ABB RobotStudio station: proyecto final.rspag

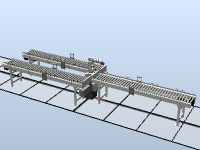
--- station ---
Station proyecto final_4 (saved by RobotStudio 6.8.8307.1040)
Controller ProyectoFinal, task T_ROB1: task frame (RAPID world) sits at (45.04, 0, 650) mm in the station
Controller ProyectoFinal
  mechanical unit ROB_1: IRB120_3_58__01, 6 joints, base frame (0, 0, 0) mm
Layout (positions relative to the parent item):
  - IRB120_3_58__01 [mechanism, from Robots\IRB120_3_58_G_01.rslib] at (45.04, 0, 650) mm; joint values [0, 0, 0, 0, 0.5236, 0] (rad or m)
  - RobotBase [part, from Descargas del Explorador\RobotBase.rslib] at (-150, -150, 0) mm
  - 400_guide [part, from Equipment\Conveyor Guide 400.rslib] at (192.48, -209.68, 0) mm
  - 400_guide_Big [part, from Equipment\Conveyor Guide 400.rslib] at (168.85, 683.15, 0) mm, rotated rx 0 ry 0 rz 180 deg
  - 400_guide_Small [part, from Equipment\Conveyor Guide 400.rslib] at (130.41, -257.14, 0) mm, rotated rx 0 ry 0 rz 180 deg
  - Big_Can [part] at (3492.94, 0, 776.65) mm
  - Little_Can [part] at (3339.79, 0, 775.69) mm
  - SmartComponent_1 [smart component]
      signals: DI Cinta1, DI Marcha, DO Sensor1Big, DO Sensor1Small, DI Cinta2Big, DI Cinta2Small, DI CogerC1Big, DI CogerC1Small, DI DejarC1Big, DI DejarC1Small, DO Sensor2Big, DO Sensor2Small, DI Cinta1S, DI Marcha1S
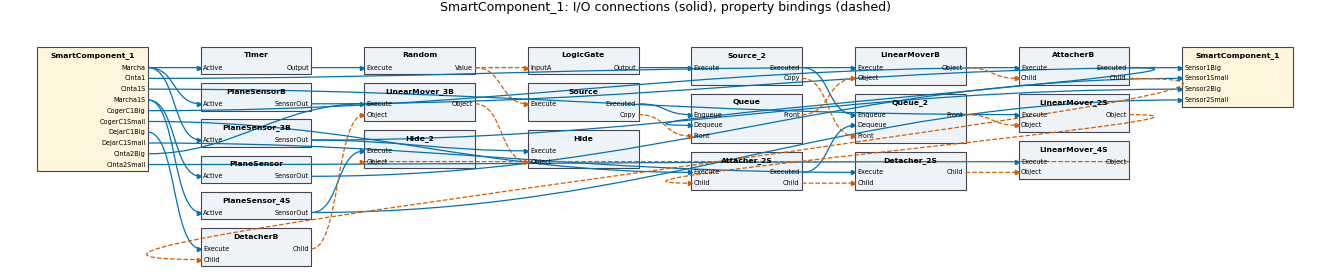
      connections:
        SmartComponent_1.Marcha -> Timer.Active
        Timer.Output -> Random.Execute
        LogicGate.Output -> Source_2.Execute
        Source.Executed -> Queue.Enqueue
        Source_2.Executed -> Queue_2.Enqueue
        SmartComponent_1.Cinta1 -> LinearMoverB.Execute
        SmartComponent_1.Cinta1S -> LinearMover_2S.Execute
        PlaneSensorB.SensorOut -> SmartComponent_1.Sensor1Big
        PlaneSensor.SensorOut -> SmartComponent_1.Sensor1Small
        SmartComponent_1.Marcha -> PlaneSensorB.Active
        SmartComponent_1.Marcha1S -> PlaneSensor.Active
        SmartComponent_1.CogerC1Big -> AttacherB.Execute
        SmartComponent_1.CogerC1Small -> Attacher_2S.Execute
        SmartComponent_1.DejarC1Big -> DetacherB.Execute
        SmartComponent_1.DejarC1Small -> Detacher_2S.Execute
        SmartComponent_1.Marcha -> PlaneSensor_3B.Active
        SmartComponent_1.Marcha1S -> PlaneSensor_4S.Active
        PlaneSensor_3B.SensorOut -> SmartComponent_1.Sensor2Big
        PlaneSensor_4S.SensorOut -> SmartComponent_1.Sensor2Small
        SmartComponent_1.Cinta2Big -> LinearMover_3B.Execute
        SmartComponent_1.Cinta2Small -> LinearMover_4S.Execute
        AttacherB.Executed -> Queue.Dequeue
        Attacher_2S.Executed -> Queue_2.Dequeue
        PlaneSensor_3B.SensorOut -> Hide.Execute
        PlaneSensor_4S.SensorOut -> Hide_2.Execute
        Random.Value => LogicGate.InputA
        Random.Value => Source.Execute
        Source.Copy => Queue.Front
        Source_2.Copy => Queue_2.Front
        Queue.Front => LinearMoverB.Object
        Queue_2.Front => LinearMover_2S.Object
        LinearMoverB.Object => AttacherB.Child
        LinearMover_2S.Object => Attacher_2S.Child
        AttacherB.Child => DetacherB.Child
        Attacher_2S.Child => Detacher_2S.Child
        DetacherB.Child => LinearMover_3B.Object
        Detacher_2S.Child => LinearMover_4S.Object
        LinearMover_3B.Object => Hide.Object
        LinearMover_4S.Object => Hide_2.Object
    - PlaneSensorB [smart component, from Components\PlaneSensor.rslib] at (395.44, -52.44, 915.91) mm, rotated rx 0 ry -90 rz 0 deg
        properties: Origin=[0 0 0]; Axis1=[0.1 0 0]; Axis2=[0 0.1 0]; SensedPart=(none)
      - _sensorPart_ [part, from Components\PlaneSensor.rslib]
    - Timer [smart component, from Components\Timer.rslib]
        properties: StartTime=0; Interval=7; Repeat=true; CurrentTime=20.088
    - Queue [smart component, from Components\Queue.rslib]
        properties: Back=(none); Front=(none); Queue=; NumberOfObjects=0
    - Queue_2 [smart component, from Components\Queue.rslib]
        properties: Back=(none); Front=(none); Queue=; NumberOfObjects=0
    - Source [smart component, from Components\Source.rslib]
        properties: Source=Big_Can; Copy=(none); Parent=(none); Position=[2.892064 0 0.776651]; Orientation=[0 0 0]; Transient=true; PhysicsBehavior=0
    - Source_2 [smart component, from Components\Source.rslib]
        properties: Source=Little_Can; Copy=(none); Parent=(none); Position=[2.753947 0 0.775688]; Orientation=[0 0 0]; Transient=true; PhysicsBehavior=0
    - LinearMoverB [smart component, from Components\LinearMover.rslib]
        properties: Object=(none); Direction=[-1 0 0]; Speed=0.8; Reference=Global; ReferenceObject=(none)
    - Random [smart component, from Components\Random.rslib]
        properties: Value=0.788703927206203; Min=0; Max=1
    - LogicGate [smart component, from Components\LogicGate.rslib]
        properties: Operator=NOT; Delay=0
    - LinearMover_2S [smart component, from Components\LinearMover.rslib]
        properties: Object=(none); Direction=[-1 0 0]; Speed=0.8; Reference=Global; ReferenceObject=(none)
    - PlaneSensor_3B [smart component, from Components\PlaneSensor.rslib] at (-2635.89, 427.82, 780.39) mm
        properties: Origin=[0 0 0]; Axis1=[0.1 0 0]; Axis2=[0 0.1 0]; SensedPart=(none)
      - _sensorPart_ [part, from Components\PlaneSensor.rslib]
    - PlaneSensor_4S [smart component, from Components\PlaneSensor.rslib] at (-2612.83, -525.9, 779.66) mm
        properties: Origin=[0 0 0]; Axis1=[0.1 0 0]; Axis2=[0 0.1 0]; SensedPart=(none)
      - _sensorPart_ [part, from Components\PlaneSensor.rslib]
    - AttacherB [smart component, from Components\Attacher.rslib]
        properties: Parent=subcionador pro; Flange=0; Child=(none); Mount=false; Offset=[0 0 0]; Orientation=[0 0 0]
    - Attacher_2S [smart component, from Components\Attacher.rslib]
        properties: Parent=subcionador pro; Flange=0; Child=(none); Mount=false; Offset=[0 0 0]; Orientation=[0 0 0]
    - DetacherB [smart component, from Components\Detacher.rslib]
        properties: Child=(none); KeepPosition=true
    - Detacher_2S [smart component, from Components\Detacher.rslib]
        properties: Child=(none); KeepPosition=true
    - LinearMover_3B [smart component, from Components\LinearMover.rslib]
        properties: Object=(none); Direction=[-1 0 0]; Speed=1.8; Reference=Global; ReferenceObject=(none)
    - LinearMover_4S [smart component, from Components\LinearMover.rslib]
        properties: Object=(none); Direction=[-1 0 0]; Speed=1.8; Reference=Global; ReferenceObject=(none)
    - PlaneSensor [smart component, from Components\PlaneSensor.rslib] at (387.44, -48.08, 820.06) mm, rotated rx 0 ry -90 rz 0 deg
        properties: Origin=[0 0 0]; Axis1=[0.1 0 0]; Axis2=[0 0.1 0]; SensedPart=(none)
      - _sensorPart_ [part, from Components\PlaneSensor.rslib]
    - Hide [smart component, from Components\Hide.rslib]
        properties: Object=(none)
    - Hide_2 [smart component, from Components\Hide.rslib]
        properties: Object=(none)
  - subcionador pro [mechanism, from Videos\subcionador pro.rslib] at (409.39, 0, 1244) mm, rotated rx 180 ry 60 rz 180 deg
Attachment: subcionador pro is attached to IRB120_3_58__01 / Link6
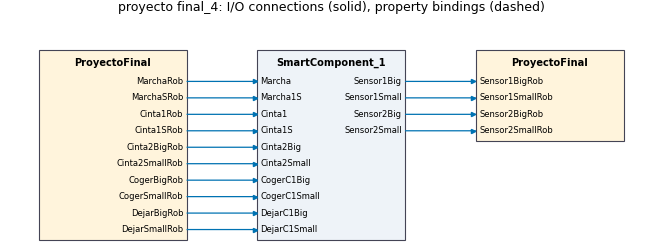
Station logic (signal -> signal, property => property):
  ProyectoFinal.MarchaRob -> SmartComponent_1.Marcha
  ProyectoFinal.MarchaSRob -> SmartComponent_1.Marcha1S
  ProyectoFinal.Cinta1Rob -> SmartComponent_1.Cinta1
  ProyectoFinal.Cinta1SRob -> SmartComponent_1.Cinta1S
  SmartComponent_1.Sensor1Big -> ProyectoFinal.Sensor1BigRob
  SmartComponent_1.Sensor1Small -> ProyectoFinal.Sensor1SmallRob
  ProyectoFinal.Cinta2BigRob -> SmartComponent_1.Cinta2Big
  ProyectoFinal.Cinta2SmallRob -> SmartComponent_1.Cinta2Small
  ProyectoFinal.CogerBigRob -> SmartComponent_1.CogerC1Big
  ProyectoFinal.CogerSmallRob -> SmartComponent_1.CogerC1Small
  ProyectoFinal.DejarBigRob -> SmartComponent_1.DejarC1Big
  ProyectoFinal.DejarSmallRob -> SmartComponent_1.DejarC1Small
  SmartComponent_1.Sensor2Big -> ProyectoFinal.Sensor2BigRob
  SmartComponent_1.Sensor2Small -> ProyectoFinal.Sensor2SmallRob
Targets, tools, work objects and paths stored in the station and not in the controller backup, written as RAPID:
! task T_ROB1
MODULE Module1
  PROC pieza()
    robotSmall;
    sensar1;
  ENDPROC
  PROC cicle()
    SetDO CogerBigRob,0;
    SetDO DejarBigRob,0;
    SetDO CogerSmallRob,0;
    SetDO DejarSmallRob,0;
    SetDO MarchaRob,1;
    SetDO MarchaSRob,1;
    SetDO Cinta1Rob,1;
    SetDO Cinta1SRob,1;
    SetDO Cinta2BigRob,0;
    SetDO Cinta2SmallRob,0;
    WaitDI Sensor1SmallRob,1;
    SetDO Cinta1Rob,0;
    SetDO Cinta1SRob,0;
    piezas;
  ENDPROC
  PROC sensar()
    cicle;
    cicle;
  ENDPROC
ENDMODULE


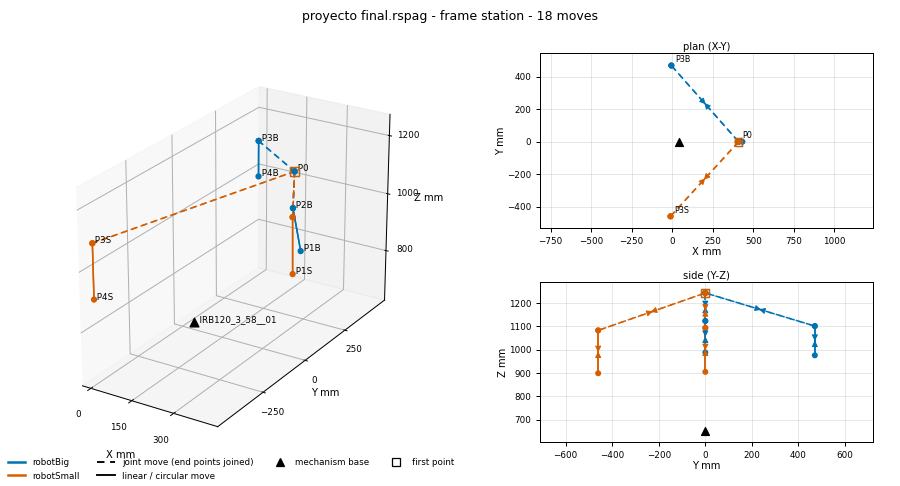
[picture p0: tool path of proyecto final.rspag in frame station, 18 of 18 moves have a stored position in this frame; points joined in program order, loops and branches not executed]
--- Backups/ProyectoFinal/RAPID/TASK1/PROGMOD/CalibData.mod ---
MODULE CalibData
ENDMODULE

--- Backups/ProyectoFinal/RAPID/TASK1/PROGMOD/Module1.mod ---
MODULE Module1
    CONST robtarget P0:=[[364.353829072,0,594],[0.5,0,0.866025404,0],[0,0,0,0],[9E+09,9E+09,9E+09,9E+09,9E+09,9E+09]];
    CONST robtarget P2B:=[[360.022653153,0,473.726196092],[0,0,1,0],[0,0,0,0],[9E+09,9E+09,9E+09,9E+09,9E+09,9E+09]];
    CONST robtarget P1B:=[[388.755601806,0,338.420809037],[0,0,1,0],[0,0,0,0],[9E+09,9E+09,9E+09,9E+09,9E+09,9E+09]];
    CONST robtarget P3B:=[[-50.206591399,470.402076052,451.620152637],[0,0,1,0],[0,0,0,0],[9E+09,9E+09,9E+09,9E+09,9E+09,9E+09]];
    CONST robtarget P4B:=[[-50.206591399,470.402076052,325.966309799],[0,0,1,0],[0,0,0,0],[9E+09,9E+09,9E+09,9E+09,9E+09,9E+09]];
    CONST robtarget P2S:=[[359.130975003,0,443.778021736],[0,0,1,0],[0,0,0,0],[9E+09,9E+09,9E+09,9E+09,9E+09,9E+09]];
    CONST robtarget P1S:=[[361.332509941,0,254.842738956],[0,0,1,0],[0,0,0,0],[9E+09,9E+09,9E+09,9E+09,9E+09,9E+09]];
    CONST robtarget P3S:=[[-55.454860484,-460.39542717,433.082453731],[0,0,1,0],[-2,0,-2,0],[9E+09,9E+09,9E+09,9E+09,9E+09,9E+09]];
    CONST robtarget P4S:=[[-55.454860484,-460.39542717,248.927934739],[0,0,1,0],[-2,0,-2,0],[9E+09,9E+09,9E+09,9E+09,9E+09,9E+09]];
	PERS tooldata subcionador_pro:=[TRUE,[[0,0,0],[1,0,0,0]],[2,[0,0,1],[1,0,0,0],0,0,0]];
    !***********************************************************
    !
    ! Module:  Module1
    !
    ! Description:
    !   <Pick and Place de dos diferentes latas>
    !
    ! Author: Kenneth
    !
    ! Version: 1.0
    !
    !***********************************************************


    !***********************************************************
    !
    ! Procedure main
    !
    !   This is the entry point of your program
    !
    !***********************************************************
    PROC main()
        !Aqui pongo las señales de agarrar y soltar las latas en 0, así cada vez que se inicia, empiezan en 0
        SetDO CogerBigRob,0;
        SetDO DejarBigRob,0;
        SetDO CogerSmallRob,0;
        SetDO DejarSmallRob,0;
        !Aquí pongo en marcha la cinta, son dos porque para evitar cualquier error hice que cada lata actuara
        !como si se movieran en cintas diferentes
        SetDO MarchaRob,1;
        SetDO MarchaSRob,1;
        SetDO Cinta1Rob,1;
        SetDO Cinta1SRob,1;
        SetDO Cinta2BigRob,0;
        SetDO Cinta2SmallRob,0;
        !Apenas el sensor que tiene contacto con los dos tipos de latas recibe una señal, para la cinta para
        !realizar la función piezas
        WaitDI Sensor1SmallRob,1;
        SetDO Cinta1Rob,0;
        SetDO Cinta1SRob,0;
        piezas;
    ENDPROC
    PROC robotBig()
        !Trayectoria para las latas grandes
        MoveJ P0,v1000,z100,subcionador_pro\WObj:=wobj0;
        MoveJ P2B,v1000,z100,subcionador_pro\WObj:=wobj0;
        MoveL P1B,v1000,fine,subcionador_pro\WObj:=wobj0;
        SetDO CogerBigRob,1;
        MoveL P2B,v1000,z100,subcionador_pro\WObj:=wobj0;
        MoveJ P0,v1000,z100,subcionador_pro\WObj:=wobj0;
        MoveJ P3B,v1000,z100,subcionador_pro\WObj:=wobj0;
        MoveL P4B,v1000,fine,subcionador_pro\WObj:=wobj0;
        SetDO DejarBigRob,1;
        SetDO Cinta2BigRob,1;
        MoveL P3B,v1000,z100,subcionador_pro\WObj:=wobj0;
        MoveJ P0,v1000,z100,subcionador_pro\WObj:=wobj0;
        WaitDI Sensor2BigRob,1;
        SetDO Cinta2BigRob,0;
        SetDO Cinta1Rob,1;
    ENDPROC
    PROC robotSmall()
        !Trayectoria para las latas chicas
        MoveJ P0,v1000,z100,subcionador_pro\WObj:=wobj0;
        MoveJ P2S,v1000,z100,subcionador_pro\WObj:=wobj0;
        MoveL P1S,v1000,fine,subcionador_pro\WObj:=wobj0;
        SetDO CogerSmallRob,1;
        MoveL P2S,v1000,z100,subcionador_pro\WObj:=wobj0;
        MoveJ P0,v1000,z100,subcionador_pro\WObj:=wobj0;
        MoveJ P3S,v1000,z100,subcionador_pro\WObj:=wobj0;
        MoveL P4S,v1000,fine,subcionador_pro\WObj:=wobj0;
        SetDO DejarSmallRob,1;
        SetDO Cinta2SmallRob,1;
        MoveL P3S,v1000,z100,subcionador_pro\WObj:=wobj0;
        MoveJ P0,v1000,z100,subcionador_pro\WObj:=wobj0;
        WaitDI Sensor2SmallRob,1;
        SetDO Cinta2SmallRob,0;
        SetDO Cinta1Rob,1;
    ENDPROC
   PROC piezas()
       !Esta función es para diferenciar cual pieza se va a agarrar
       !Si los dos sensores son activados se ejecuta la función robotBig, que es de la trayectoria de las
       !latas grandes y sensar2 que es para poner los valores en su forma inicial y poder tener un ciclo
       IF Sensor1SmallRob=1 AND Sensor1BigRob=1 THEN
           robotBig;
           sensar2;
        !Si solo se activa un sensor se ejecuta la función robotSmall, que es de la trayectoria de las latas
        !pequeñas y sensar1 que es para poner los valores en su forma inicial y poder tener un ciclo
        ELSEIF Sensor1SmallRob=1 AND Sensor1BigRob=0 THEN
            robotSmall;
            sensar1;
       ENDIF
    ENDPROC
   PROC sensar1()
       !si es activado el sensor final de la cinta de latas chicas se ejecuta
       !nuevamente el main
    IF Sensor2SmallRob=1 THEN
            main;
    ENDIF
   ENDPROC
   PROC sensar2()
       !si es activado el sensor final de la cinta de latas grandes se ejecuta
       !nuevamente el main
    IF Sensor2BigRob=1 THEN
            main;
    ENDIF
   ENDPROC
ENDMODULE

--- Backups/ProyectoFinal/SYSPAR/EIO.cfg ---
EIO:CFG_1.0:6:1::
#
EIO_SIGNAL:

      -Name "MarchaRob" -SignalType "DO"

      -Name "Cinta1Rob" -SignalType "DO"

      -Name "Sensor1BigRob" -SignalType "DI"

      -Name "Sensor1SmallRob" -SignalType "DI"

      -Name "Cinta2BigRob" -SignalType "DO"

      -Name "Cinta2SmallRob" -SignalType "DO"

      -Name "CogerBigRob" -SignalType "DO"

      -Name "CogerSmallRob" -SignalType "DO"

      -Name "DejarBigRob" -SignalType "DO"

      -Name "DejarSmallRob" -SignalType "DO"

      -Name "Sensor2BigRob" -SignalType "DI"

      -Name "Sensor2SmallRob" -SignalType "DI"

      -Name "Cinta1SRob" -SignalType "DO"

      -Name "MarchaSRob" -SignalType "DO"
